Universal Robots PolyScope program: barreraVirtualCub.urp

Program barreraVirtualCubPROVA (installation=default directory=/programs/usbdisk_1/provesTFGMireia/provesGithub createdIn=5.15.1.0 lastSavedIn=5.12.1.1101497 robotSerialNumber=20225300640)
Calibrated DH parameters: a=[-0.000125, -0.240482, -0.204397, 0.000169, -0.000135, 0]; d=[0.152056, 4.760815, 12.138494, -16.768367, 0.085457, 0.092357]; alpha=[1.570863, 0.008548, 0.003635, 1.571424, -1.571918, 0]; deltaTheta=[0, 0.167622, 0.124346, -0.291972, 0.000034, 0]
InitVariablesNode
Robot Program (runOnlyOnce=true)
  'Definim les variables surtTCP, surtToolFlange i surtMig com a False per indicar quin surt.'
  surtTCP := False
  surtToolFlange := False
  surtMig := False
  'Donem valor a la varialbe retrocedir.'
  retrocedir := 0.005
  'Definim els radis de les esferes del TCP, el toolFlange i el punt mig.'
  radiTCP := 0.05
  radiFlange := 0.06
  radiMig := 0.05
  'Agafem els dos punts necessaris per fer un cub perfecte.'
  p1 := p[0.150,-0.483,0.473,0,0,0]
  p2 := p[-0.149,-0.244,0.043,0,0,0]
  'Calculem el punt central.'
  centre := p[(p1[0]+p2[0])/2,(p1[1]+p2[1])/2,(p1[2]+p2[2])/2,0,0,0]
  'Activem el moviment lliure.'
  Script: freedrive_mode()
  Loop Forever
    'Surt el TCP, el Flange o el punt mig.'
    If surtTCP≟ True (checkContinuously=true)
      'Aturem el moviment lliure.'
      Script: end_freedrive_mode()
      'Obtenim la posicio actual del TCP.'
      posAct := get_actual_tcp_pose()
      'Cridem el subprograma per rectificar la posicio.'
      Call rectificarPosicio
      'Retornem les variables a False i reactivem el moviment lliure.'
      surtTCP := False
    If surtToolFlange≟ True (checkContinuously=true)
      'Aturem el moviment lliure.'
      Script: end_freedrive_mode()
      'Obtenim la posicio actual de la brida del robot.'
      posAct := get_actual_tool_flange_pose()
      'Cridem el subprograma per rectificar la posicio.'
      Call rectificarPosicio
      'Retornem les variables a False i reactivem el moviment lliure.'
      surtToolFlange := False
    If surtMig≟ True (checkContinuously=true)
      'Aturem el moviment lliure.'
      Script: end_freedrive_mode()
      'Obtenim les posicions actuals de la brida i el TCP per calcular el punt del mig.'
      tcpAct := get_actual_tcp_pose()
      flangeAct := get_actual_tool_flange_pose()
      posAct := p[(tcpAct[0]+flangeAct[0])/2,(tcpAct[1]+flangeAct[1])/2,(tcpAct[2]+flangeAct[2])/2,tcpAct[3],tcpAct[4],tcpAct[5]]
      'Cridem el subprograma per rectificar la posicio.'
      Call rectificarPosicio
      'Retornem les variables a False i reactivem el moviment lliure.'
      surtMig := False
    Wait Sleep waitTime=0.01
SubProgram -> rectificarPosicio
Thread Thread_1 (runOnlyOnce=false)
  Loop Forever
    'Obtenim les posicions del TCP, el toolFlange i el punt del mig.'
    llistaPosTCP := get_actual_tcp_pose()
    llistaPosFlange := get_actual_tool_flange_pose()
    llistaPosMig := p[(llistaPosTCP[0]+llistaPosFlange[0])/2,(llistaPosTCP[1]+llistaPosFlange[1])/2,(llistaPosTCP[2]+llistaPosFlange[2])/2,llistaPosTCP[3],llistaPosTCP[4],llistaPosTCP[5]]
    posX := llistaPosTCP[0]
    posXf := llistaPosFlange[0]
    posXm := llistaPosMig[0]
    posY := llistaPosTCP[1]
    posYf := llistaPosFlange[1]
    posYm := llistaPosMig[1]
    posZ := llistaPosTCP[2]
    posZf := llistaPosFlange[2]
    posZm := llistaPosMig[2]
    'Comprovem eixos X'
    If posX≥(p1[0]-radiTCP) or posX≤(p2[0]+radiTCP) (checkContinuously=true)
      surtTCP := True
    If posXf≥(p1[0]-radiFlange) or posXf≤(p2[0]+radiFlange) (checkContinuously=true)
      surtToolFlange := True
    If posXm≥(p1[0]-radiMig) or posXm≤(p2[0]+radiMig) (checkContinuously=true)
      surtMig := True
    'Comprovem eixos Y'
    If posY≤(p1[1]+radiTCP) or posY≥(p2[1]-radiTCP) (checkContinuously=true)
      surtTCP := True
    If posYf≤(p1[1]+radiFlange) or posYf≥(p2[1]-radiFlange) (checkContinuously=true)
      surtToolFlange := True
    If posYm≤(p1[1]+radiMig) or posYm≥(p2[1]-radiMig) (checkContinuously=true)
      surtMig := True
    'Comprovem eixos Z'
    If posZ≥(p1[2]-radiTCP) or posZ≤(p2[2]+radiTCP) (checkContinuously=true)
      surtTCP := True
    If posZf≥(p1[2]-radiFlange) or posZf≤(p2[2]+radiFlange) (checkContinuously=true)
      surtToolFlange := True
    If posZm≥(p1[2]-radiMig) or posZm≤(p2[2]+radiMig) (checkContinuously=true)
      surtMig := True
SubProgram rectificarPosicio (keepSynchronizedWithDisk=false)
  'Subprograma cridat per tal de fer un moviment amb una direccio.'
  'Abans de cridar el subprograma s'ha d'haver obtingut el valor de la posicio actual.'
  'Generem el vector director del punt actual al centre.'
  vectorDir := [centre[0]-posAct[0],centre[1]-posAct[1],centre[2]-posAct[2]]
  'Ens movem en direccio el centre fins que s'hagi recorregut una distancia determinada.'
  MoveL speed 20 mm/s, acceleration 120 mm/s^2 (useActiveTCP=true) feature=Base
    MoveDirectionNode expression=vectorDir
      Until DISTANCE (allowActions=false deceleration=3 distanceNodeType=STOP) Distance=0.005; motionParameters(blendRadius=0)
  'Tornem a activar el moviment lliure.'
  Script: freedrive_mode()
